DATA_BLOCK "呼梯管理_DB"
{ S7_Optimized_Access := 'TRUE' }
VERSION : 0.1
NON_RETAIN
"呼梯管理"

BEGIN

END_DATA_BLOCK

